FUNCTION_BLOCK FB_Opcpa_Test EXTENDS FB_TestSuite
VAR_INPUT
END_VAR
VAR_OUTPUT
END_VAR
VAR
END_VAR

END_FUNCTION_BLOCK

(* stored: Version 1.1.0.1, ProductVersion 3.1.4020.14
   POU FB_Opcpa_Test: Id {09b0b164-c94c-4024-9b95-134904e8d427}, SpecialFunc None *)
